# EPICS substitutions: elveFlowESmobileApp/Db/pid_slow.substitutions
file "$(STD)/db/pid_control.db"
{
pattern
{P,                          PID,     INP,                                    OUT,                              LOPR,  HOPR,  DRVL,  DRVH,  PREC,   KP,  KI,   KD,    SCAN}
{elveFlowOB1:,                PID1,    "XF11ID-ES\{elveFlowOB1\}:elveFlow:Sensor1_RBV",  "XF11ID-ES\{elveFlowOB1\}:elveFlow:Pres1",   0,     5,    0,     2000,    5,      0.2,  0.,   0.,  ".1 second"}
}
